{attribute 'GeneratedUsingTerminal: EK1100-0000-0018'}
{attribute addProperty BoxType "EK1100-0000-0018"}
{attribute addProperty Id "Beckhoff_EL32xxEK1122Beckhoff_EL32xxEK1122_86F9EED92A_0001_EL3201_0000_0016EL3201_771154E121A_0002_EL3201_0000_0017EL3201_F37BFE8521A_0003_EL3201_0000_0018EL3201_F37BFE8521A_0004_EL3201_0000_0019EL3201_F37BFE8521A_0005_EL3201_0000_0020EL3201_F37BFE8521A_0006_EL3201_0000_0021EL3201_F37BFE8521A_0007_EL3201_0000_0022EL3201_F37BFE8521A_0008_EL3201_0010_0016EL3201_771154E121A_0009_EL3201_0010_0017EL3201_F37BFE8521A_0010_EL3201_0010_0018EL3201_F37BFE8521A_0011_EL3201_0010_0019EL3201_F37BFE8521A_0012_EL3201_0010_0020EL3201_F37BFE8521A_0013_EL3201_0010_0021EL3201_F37BFE8521A_0014_EL3201_0010_0022EL3201_F37BFE8521A_0015_EL3201_0020_0016EL3201_771154E121A_0016_EL3201_0020_0017EL3201_F37BFE8521A_0017_EL3201_0020_0018EL3201_F37BFE8521A_0018_EL3201_0020_0019EL3201_F37BFE8521A_0019_EL3201_0020_0020EL3201_F37BFE8521A_0020_EL3201_0020_0021EL3201_F37BFE8521A_0021_EL3201_0020_0022EL3201_F37BFE8521A_0022_EL3202_0000_0016EL3202_75835C5C30A_0023_EL3202_0000_0017EL3202_27F1223730A_0024_EL3202_0000_0018EL3202_27F1223730A_0025_EL3202_0000_0019EL3202_27F1223730A_0026_EL3202_0000_0020EL3202_27F1223730A_0027_EL3202_0000_0021EL3202_27F1223730A_0028_EL3202_0000_0022EL3202_27F1223730A_0029_EL3202_0010_0016EL3202_75835C5C30A_0030_EL3202_0010_0017EL3202_27F1223730A_0031_EL3202_0010_0018EL3202_27F1223730A_0032_EL3202_0010_0019EL3202_27F1223730A_0033_EL3202_0010_0020EL3202_27F1223730A_0034_EL3202_0010_0021EL3202_27F1223730A_0035_EL3202_0010_0022EL3202_27F1223730A_0036_EL3202_0020_0017EL3202_27F1223730A_0037_EL3202_0020_0018EL3202_27F1223730A_0038_EL3202_0020_0019EL3202_27F1223730A_0039_EL3202_0020_0020EL3202_27F1223730A_0040_EL3202_0020_0021EL3202_27F1223730A_0041_EL3202_0020_0022EL3202_27F1223730A_0042_EL3204_0000_0016EL3204_6F0438BE48A_0043_EL3204_0000_0017EL3204_B6248F5B48A_0044_EL3204_0000_0018EL3204_B6248F5B48A_0045_EL3204_0000_0019EL3204_B6248F5B48A_0046_EL3204_0000_0020EL3204_B6248F5B48A_0047_EL3204_0000_0021EL3204_B6248F5B48A_0048_EL3204_0162_0016EL3204_988CC22448A_0049_EL3204_0162_0017EL3204_988CC22448A_0050_EL3204_0162_0018EL3204_988CC22448A_0051_EL3204_0162_0019EL3204_988CC22448A_0052_EL3204_0200_0016EL3204_8BBE23EA40A_0053_EL3204_0200_0017EL3204_8BBE23EA40A_0054_EL3204_0200_0018EL3204_8BBE23EA40A_0055_EL3208_0000_0017EL3208_E885804F68A_0056_EL3208_0000_0018EL3208_E885804F68A_0057_EL3208_0010_0016EL3208_E885804F68A_0058_EL3214_0000_0016EL3214_8BBE23EA40A_0059_EL3214_0000_0017EL3214_8BBE23EA40A_0060_EL3214_0090_0016EL3214_8BBE23EA40A_0061_EL3218_0000_0016EL3218_E885804F68A_0062_EL3218_0000_0017EL3218_E885804F68A_0063_EL3255_0000_0016EL3255_7067083162A_0064_EL3255_0000_0017EL3255_1972F7C062A_0065_EL3255_0000_0018EL3255_1972F7C062A_0066_EL3255_0000_0019EL3255_1972F7C062A_0067_EL3255_0000_0020EL3255_B4D4BD5144A_0068_EL3255_0000_0021EL3255_1972F7C062A_0069_EL3255_0000_0022EL3255_1972F7C062A_0070_EL3255_0000_0023EL3255_1972F7C062"}
{attribute addProperty CRC "2837355841"}
{attribute addProperty Size "2581"}
TYPE Beckhoff_EL32xx_A91E9D41 EXTENDS EK1100_1FC0878B :
STRUCT
	{attribute addProperty Name "Beckhoff_EL32xxEK1122"}
	{attribute addProperty PreviousPort "Beckhoff EL32xx : B"}
	Beckhoff_EL32xxEK1122 : Beckhoff_EL32xxEK1122_86F9EED9;
	{attribute addProperty Name "A_0001_EL3201_0000_0016"}
	{attribute addProperty PreviousPort "Beckhoff EL32xxEK1122 : C"}
	A_0001_EL3201_0000_0016 : EL3201_771154E1;
	{attribute addProperty Name "A_0002_EL3201_0000_0017"}
	{attribute addProperty PreviousPort "A_0001(EL3201-0000-0016) : B"}
	A_0002_EL3201_0000_0017 : EL3201_F37BFE85;
	{attribute addProperty Name "A_0003_EL3201_0000_0018"}
	{attribute addProperty PreviousPort "A_0002(EL3201-0000-0017) : B"}
	A_0003_EL3201_0000_0018 : EL3201_F37BFE85;
	{attribute addProperty Name "A_0004_EL3201_0000_0019"}
	{attribute addProperty PreviousPort "A_0003(EL3201-0000-0018) : B"}
	A_0004_EL3201_0000_0019 : EL3201_F37BFE85;
	{attribute addProperty Name "A_0005_EL3201_0000_0020"}
	{attribute addProperty PreviousPort "A_0004(EL3201-0000-0019) : B"}
	A_0005_EL3201_0000_0020 : EL3201_F37BFE85;
	{attribute addProperty Name "A_0006_EL3201_0000_0021"}
	{attribute addProperty PreviousPort "A_0005(EL3201-0000-0020) : B"}
	A_0006_EL3201_0000_0021 : EL3201_F37BFE85;
	{attribute addProperty Name "A_0007_EL3201_0000_0022"}
	{attribute addProperty PreviousPort "A_0006(EL3201-0000-0021) : B"}
	A_0007_EL3201_0000_0022 : EL3201_F37BFE85;
	{attribute addProperty Name "A_0008_EL3201_0010_0016"}
	{attribute addProperty PreviousPort "A_0007(EL3201-0000-0022) : B"}
	A_0008_EL3201_0010_0016 : EL3201_771154E1;
	{attribute addProperty Name "A_0009_EL3201_0010_0017"}
	{attribute addProperty PreviousPort "A_0008(EL3201-0010-0016) : B"}
	A_0009_EL3201_0010_0017 : EL3201_F37BFE85;
	{attribute addProperty Name "A_0010_EL3201_0010_0018"}
	{attribute addProperty PreviousPort "A_0009(EL3201-0010-0017) : B"}
	A_0010_EL3201_0010_0018 : EL3201_F37BFE85;
	{attribute addProperty Name "A_0011_EL3201_0010_0019"}
	{attribute addProperty PreviousPort "A_0010(EL3201-0010-0018) : B"}
	A_0011_EL3201_0010_0019 : EL3201_F37BFE85;
	{attribute addProperty Name "A_0012_EL3201_0010_0020"}
	{attribute addProperty PreviousPort "A_0011(EL3201-0010-0019) : B"}
	A_0012_EL3201_0010_0020 : EL3201_F37BFE85;
	{attribute addProperty Name "A_0013_EL3201_0010_0021"}
	{attribute addProperty PreviousPort "A_0012(EL3201-0010-0020) : B"}
	A_0013_EL3201_0010_0021 : EL3201_F37BFE85;
	{attribute addProperty Name "A_0014_EL3201_0010_0022"}
	{attribute addProperty PreviousPort "A_0013(EL3201-0010-0021) : B"}
	A_0014_EL3201_0010_0022 : EL3201_F37BFE85;
	{attribute addProperty Name "A_0015_EL3201_0020_0016"}
	{attribute addProperty PreviousPort "A_0014(EL3201-0010-0022) : B"}
	A_0015_EL3201_0020_0016 : EL3201_771154E1;
	{attribute addProperty Name "A_0016_EL3201_0020_0017"}
	{attribute addProperty PreviousPort "A_0015(EL3201-0020-0016) : B"}
	A_0016_EL3201_0020_0017 : EL3201_F37BFE85;
	{attribute addProperty Name "A_0017_EL3201_0020_0018"}
	{attribute addProperty PreviousPort "A_0016(EL3201-0020-0017) : B"}
	A_0017_EL3201_0020_0018 : EL3201_F37BFE85;
	{attribute addProperty Name "A_0018_EL3201_0020_0019"}
	{attribute addProperty PreviousPort "A_0017(EL3201-0020-0018) : B"}
	A_0018_EL3201_0020_0019 : EL3201_F37BFE85;
	{attribute addProperty Name "A_0019_EL3201_0020_0020"}
	{attribute addProperty PreviousPort "A_0018(EL3201-0020-0019) : B"}
	A_0019_EL3201_0020_0020 : EL3201_F37BFE85;
	{attribute addProperty Name "A_0020_EL3201_0020_0021"}
	{attribute addProperty PreviousPort "A_0019(EL3201-0020-0020) : B"}
	A_0020_EL3201_0020_0021 : EL3201_F37BFE85;
	{attribute addProperty Name "A_0021_EL3201_0020_0022"}
	{attribute addProperty PreviousPort "A_0020(EL3201-0020-0021) : B"}
	A_0021_EL3201_0020_0022 : EL3201_F37BFE85;
	{attribute addProperty Name "A_0022_EL3202_0000_0016"}
	{attribute addProperty PreviousPort "A_0021(EL3201-0020-0022) : B"}
	A_0022_EL3202_0000_0016 : EL3202_75835C5C;
	{attribute addProperty Name "A_0023_EL3202_0000_0017"}
	{attribute addProperty PreviousPort "A_0022(EL3202-0000-0016) : B"}
	A_0023_EL3202_0000_0017 : EL3202_27F12237;
	{attribute addProperty Name "A_0024_EL3202_0000_0018"}
	{attribute addProperty PreviousPort "A_0023(EL3202-0000-0017) : B"}
	A_0024_EL3202_0000_0018 : EL3202_27F12237;
	{attribute addProperty Name "A_0025_EL3202_0000_0019"}
	{attribute addProperty PreviousPort "A_0024(EL3202-0000-0018) : B"}
	A_0025_EL3202_0000_0019 : EL3202_27F12237;
	{attribute addProperty Name "A_0026_EL3202_0000_0020"}
	{attribute addProperty PreviousPort "A_0025(EL3202-0000-0019) : B"}
	A_0026_EL3202_0000_0020 : EL3202_27F12237;
	{attribute addProperty Name "A_0027_EL3202_0000_0021"}
	{attribute addProperty PreviousPort "A_0026(EL3202-0000-0020) : B"}
	A_0027_EL3202_0000_0021 : EL3202_27F12237;
	{attribute addProperty Name "A_0028_EL3202_0000_0022"}
	{attribute addProperty PreviousPort "A_0027(EL3202-0000-0021) : B"}
	A_0028_EL3202_0000_0022 : EL3202_27F12237;
	{attribute addProperty Name "A_0029_EL3202_0010_0016"}
	{attribute addProperty PreviousPort "A_0028(EL3202-0000-0022) : B"}
	A_0029_EL3202_0010_0016 : EL3202_75835C5C;
	{attribute addProperty Name "A_0030_EL3202_0010_0017"}
	{attribute addProperty PreviousPort "A_0029(EL3202-0010-0016) : B"}
	A_0030_EL3202_0010_0017 : EL3202_27F12237;
	{attribute addProperty Name "A_0031_EL3202_0010_0018"}
	{attribute addProperty PreviousPort "A_0030(EL3202-0010-0017) : B"}
	A_0031_EL3202_0010_0018 : EL3202_27F12237;
	{attribute addProperty Name "A_0032_EL3202_0010_0019"}
	{attribute addProperty PreviousPort "A_0031(EL3202-0010-0018) : B"}
	A_0032_EL3202_0010_0019 : EL3202_27F12237;
	{attribute addProperty Name "A_0033_EL3202_0010_0020"}
	{attribute addProperty PreviousPort "A_0032(EL3202-0010-0019) : B"}
	A_0033_EL3202_0010_0020 : EL3202_27F12237;
	{attribute addProperty Name "A_0034_EL3202_0010_0021"}
	{attribute addProperty PreviousPort "A_0033(EL3202-0010-0020) : B"}
	A_0034_EL3202_0010_0021 : EL3202_27F12237;
	{attribute addProperty Name "A_0035_EL3202_0010_0022"}
	{attribute addProperty PreviousPort "A_0034(EL3202-0010-0021) : B"}
	A_0035_EL3202_0010_0022 : EL3202_27F12237;
	{attribute addProperty Name "A_0036_EL3202_0020_0017"}
	{attribute addProperty PreviousPort "A_0035(EL3202-0010-0022) : B"}
	A_0036_EL3202_0020_0017 : EL3202_27F12237;
	{attribute addProperty Name "A_0037_EL3202_0020_0018"}
	{attribute addProperty PreviousPort "A_0036(EL3202-0020-0017) : B"}
	A_0037_EL3202_0020_0018 : EL3202_27F12237;
	{attribute addProperty Name "A_0038_EL3202_0020_0019"}
	{attribute addProperty PreviousPort "A_0037(EL3202-0020-0018) : B"}
	A_0038_EL3202_0020_0019 : EL3202_27F12237;
	{attribute addProperty Name "A_0039_EL3202_0020_0020"}
	{attribute addProperty PreviousPort "A_0038(EL3202-0020-0019) : B"}
	A_0039_EL3202_0020_0020 : EL3202_27F12237;
	{attribute addProperty Name "A_0040_EL3202_0020_0021"}
	{attribute addProperty PreviousPort "A_0039(EL3202-0020-0020) : B"}
	A_0040_EL3202_0020_0021 : EL3202_27F12237;
	{attribute addProperty Name "A_0041_EL3202_0020_0022"}
	{attribute addProperty PreviousPort "A_0040(EL3202-0020-0021) : B"}
	A_0041_EL3202_0020_0022 : EL3202_27F12237;
	{attribute addProperty Name "A_0042_EL3204_0000_0016"}
	{attribute addProperty PreviousPort "A_0041(EL3202-0020-0022) : B"}
	A_0042_EL3204_0000_0016 : EL3204_6F0438BE;
	{attribute addProperty Name "A_0043_EL3204_0000_0017"}
	{attribute addProperty PreviousPort "A_0042(EL3204-0000-0016) : B"}
	A_0043_EL3204_0000_0017 : EL3204_B6248F5B;
	{attribute addProperty Name "A_0044_EL3204_0000_0018"}
	{attribute addProperty PreviousPort "A_0043(EL3204-0000-0017) : B"}
	A_0044_EL3204_0000_0018 : EL3204_B6248F5B;
	{attribute addProperty Name "A_0045_EL3204_0000_0019"}
	{attribute addProperty PreviousPort "A_0044(EL3204-0000-0018) : B"}
	A_0045_EL3204_0000_0019 : EL3204_B6248F5B;
	{attribute addProperty Name "A_0046_EL3204_0000_0020"}
	{attribute addProperty PreviousPort "A_0045(EL3204-0000-0019) : B"}
	A_0046_EL3204_0000_0020 : EL3204_B6248F5B;
	{attribute addProperty Name "A_0047_EL3204_0000_0021"}
	{attribute addProperty PreviousPort "A_0046(EL3204-0000-0020) : B"}
	A_0047_EL3204_0000_0021 : EL3204_B6248F5B;
	{attribute addProperty Name "A_0048_EL3204_0162_0016"}
	{attribute addProperty PreviousPort "A_0047(EL3204-0000-0021) : B"}
	A_0048_EL3204_0162_0016 : EL3204_988CC224;
	{attribute addProperty Name "A_0049_EL3204_0162_0017"}
	{attribute addProperty PreviousPort "A_0048(EL3204-0162-0016) : B"}
	A_0049_EL3204_0162_0017 : EL3204_988CC224;
	{attribute addProperty Name "A_0050_EL3204_0162_0018"}
	{attribute addProperty PreviousPort "A_0049(EL3204-0162-0017) : B"}
	A_0050_EL3204_0162_0018 : EL3204_988CC224;
	{attribute addProperty Name "A_0051_EL3204_0162_0019"}
	{attribute addProperty PreviousPort "A_0050(EL3204-0162-0018) : B"}
	A_0051_EL3204_0162_0019 : EL3204_988CC224;
	{attribute addProperty Name "A_0052_EL3204_0200_0016"}
	{attribute addProperty PreviousPort "A_0051(EL3204-0162-0019) : B"}
	A_0052_EL3204_0200_0016 : EL3204_8BBE23EA;
	{attribute addProperty Name "A_0053_EL3204_0200_0017"}
	{attribute addProperty PreviousPort "A_0052(EL3204-0200-0016) : B"}
	A_0053_EL3204_0200_0017 : EL3204_8BBE23EA;
	{attribute addProperty Name "A_0054_EL3204_0200_0018"}
	{attribute addProperty PreviousPort "A_0053(EL3204-0200-0017) : B"}
	A_0054_EL3204_0200_0018 : EL3204_8BBE23EA;
	{attribute addProperty Name "A_0055_EL3208_0000_0017"}
	{attribute addProperty PreviousPort "A_0054(EL3204-0200-0018) : B"}
	A_0055_EL3208_0000_0017 : EL3208_E885804F;
	{attribute addProperty Name "A_0056_EL3208_0000_0018"}
	{attribute addProperty PreviousPort "A_0055(EL3208-0000-0017) : B"}
	A_0056_EL3208_0000_0018 : EL3208_E885804F;
	{attribute addProperty Name "A_0057_EL3208_0010_0016"}
	{attribute addProperty PreviousPort "A_0056(EL3208-0000-0018) : B"}
	A_0057_EL3208_0010_0016 : EL3208_E885804F;
	{attribute addProperty Name "A_0058_EL3214_0000_0016"}
	{attribute addProperty PreviousPort "A_0057(EL3208-0010-0016) : B"}
	A_0058_EL3214_0000_0016 : EL3214_8BBE23EA;
	{attribute addProperty Name "A_0059_EL3214_0000_0017"}
	{attribute addProperty PreviousPort "A_0058(EL3214-0000-0016) : B"}
	A_0059_EL3214_0000_0017 : EL3214_8BBE23EA;
	{attribute addProperty Name "A_0060_EL3214_0090_0016"}
	{attribute addProperty PreviousPort "A_0059(EL3214-0000-0017) : B"}
	A_0060_EL3214_0090_0016 : EL3214_8BBE23EA;
	{attribute addProperty Name "A_0061_EL3218_0000_0016"}
	{attribute addProperty PreviousPort "A_0060(EL3214-0090-0016) : B"}
	A_0061_EL3218_0000_0016 : EL3218_E885804F;
	{attribute addProperty Name "A_0062_EL3218_0000_0017"}
	{attribute addProperty PreviousPort "A_0061(EL3218-0000-0016) : B"}
	A_0062_EL3218_0000_0017 : EL3218_E885804F;
	{attribute addProperty Name "A_0063_EL3255_0000_0016"}
	{attribute addProperty PreviousPort "A_0062(EL3218-0000-0017) : B"}
	A_0063_EL3255_0000_0016 : EL3255_70670831;
	{attribute addProperty Name "A_0064_EL3255_0000_0017"}
	{attribute addProperty PreviousPort "A_0063(EL3255-0000-0016) : B"}
	A_0064_EL3255_0000_0017 : EL3255_1972F7C0;
	{attribute addProperty Name "A_0065_EL3255_0000_0018"}
	{attribute addProperty PreviousPort "A_0064(EL3255-0000-0017) : B"}
	A_0065_EL3255_0000_0018 : EL3255_1972F7C0;
	{attribute addProperty Name "A_0066_EL3255_0000_0019"}
	{attribute addProperty PreviousPort "A_0065(EL3255-0000-0018) : B"}
	A_0066_EL3255_0000_0019 : EL3255_1972F7C0;
	{attribute addProperty Name "A_0067_EL3255_0000_0020"}
	{attribute addProperty PreviousPort "A_0066(EL3255-0000-0019) : B"}
	A_0067_EL3255_0000_0020 : EL3255_B4D4BD51;
	{attribute addProperty Name "A_0068_EL3255_0000_0021"}
	{attribute addProperty PreviousPort "A_0067(EL3255-0000-0020) : B"}
	A_0068_EL3255_0000_0021 : EL3255_1972F7C0;
	{attribute addProperty Name "A_0069_EL3255_0000_0022"}
	{attribute addProperty PreviousPort "A_0068(EL3255-0000-0021) : B"}
	A_0069_EL3255_0000_0022 : EL3255_1972F7C0;
	{attribute addProperty Name "A_0070_EL3255_0000_0023"}
	{attribute addProperty PreviousPort "A_0069(EL3255-0000-0022) : B"}
	A_0070_EL3255_0000_0023 : EL3255_1972F7C0;
END_STRUCT
END_TYPE

(* stored: Version 1.2.0.0, ProductVersion 3.1.4024.9
   DUT Beckhoff_EL32xx_A91E9D41: Id {4e238414-c5c9-41d0-85a9-8321eb48aacd} *)
